PROGRAM MAIN
VAR
END_VAR

END_PROGRAM

(* stored: Version 1.1.0.1, ProductVersion 3.1.0.36
   POU MAIN: Id {e7641381-a5f8-4a6f-beee-ff3c74213a0a} *)
